// SIMATIC S7-200 SMART project (STEP 7-Micro/WIN SMART), CPU ST20

SYMBOL_TABLE 系统符号
Always_On        SM0.0    // 始终接通
END_SYMBOL_TABLE

ORGANIZATION_BLOCK MAIN:OB1
TITLE=程序注释
BEGIN
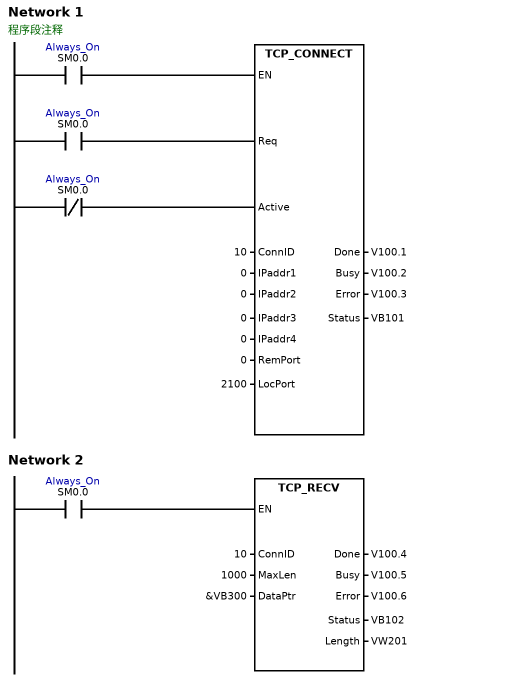
Network 1
// 程序段注释
LD     Always_On:SM0.0
=      L60.0
LD     Always_On:SM0.0
=      L63.7
LDN    Always_On:SM0.0
=      L63.6
LD     L60.0
CALL   TCP_CONNECT:SBR1, L63.7, L63.6, 10, 0, 0, 0, 0, 0, 2100, V100.1, V100.2, V100.3, VB101
Network 2
LD     Always_On:SM0.0
CALL   TCP_RECV:SBR2, 10, 1000, &VB300, V100.4, V100.5, V100.6, VB102, VW201
END_ORGANIZATION_BLOCK

// SBR1: protected block, not included

// SBR2: protected block, not included
